FUNCTION_BLOCK AO1 (* Composite Function Block Type *)
  (* Standard: 61499-2 *)
  (* Version 0.0, 2018-12-26, 4DIAC-IDE, 4DIAC-Consortium *)
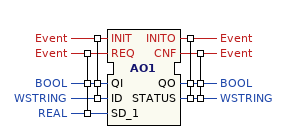
  EVENT_INPUT
    INIT WITH QI, ID; (* Initialization Request *)
    REQ WITH SD_1, QI; (* Normal Execution Request *)
  END_EVENT
  EVENT_OUTPUT
    INITO WITH QO, STATUS; (* Initialization Confirm *)
    CNF WITH QO, STATUS; (* Execution Confirmation *)
  END_EVENT
  VAR_INPUT
    QI : BOOL;
    ID : WSTRING;
    SD_1 : REAL;
  END_VAR
  VAR_OUTPUT
    QO : BOOL;
    STATUS : WSTRING;
  END_VAR
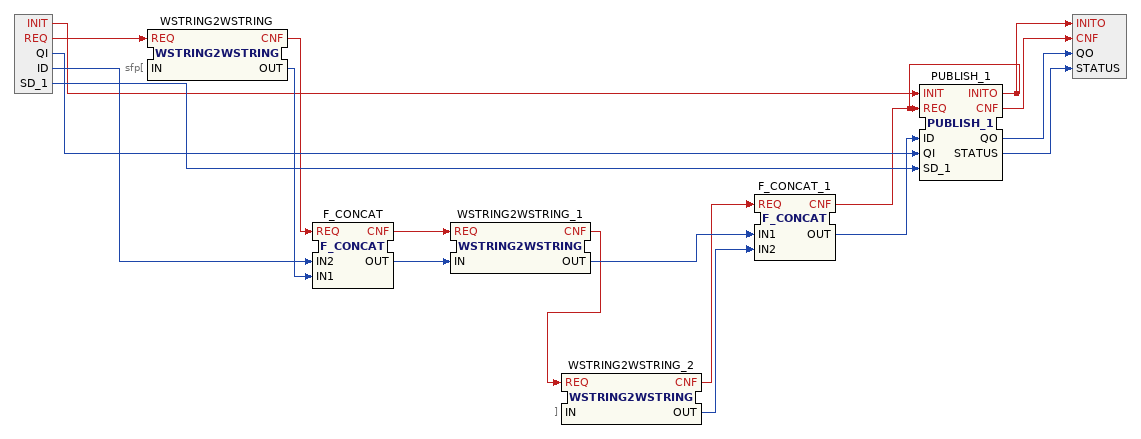
  FBS
    PUBLISH_1 : PUBLISH_1;
    F_CONCAT : F_CONCAT;
    WSTRING2WSTRING : WSTRING2WSTRING(IN := sfp[);
    WSTRING2WSTRING_1 : WSTRING2WSTRING;
    F_CONCAT_1 : F_CONCAT;
    WSTRING2WSTRING_2 : WSTRING2WSTRING(IN := ]);
  END_FBS
  EVENT_CONNECTIONS
    INIT TO PUBLISH_1.INIT;
    REQ TO WSTRING2WSTRING.REQ;
    WSTRING2WSTRING.CNF TO F_CONCAT.REQ;
    F_CONCAT.CNF TO WSTRING2WSTRING_1.REQ;
    WSTRING2WSTRING_2.CNF TO F_CONCAT_1.REQ;
    WSTRING2WSTRING_1.CNF TO WSTRING2WSTRING_2.REQ;
    F_CONCAT_1.CNF TO PUBLISH_1.REQ;
    PUBLISH_1.INITO TO INITO;
    PUBLISH_1.CNF TO CNF;
    PUBLISH_1.INITO TO PUBLISH_1.REQ;
  END_CONNECTIONS
  DATA_CONNECTIONS
    ID TO F_CONCAT.IN2;
    WSTRING2WSTRING.OUT TO F_CONCAT.IN1;
    F_CONCAT.OUT TO WSTRING2WSTRING_1.IN;
    WSTRING2WSTRING_1.OUT TO F_CONCAT_1.IN1;
    WSTRING2WSTRING_2.OUT TO F_CONCAT_1.IN2;
    F_CONCAT_1.OUT TO PUBLISH_1.ID;
    QI TO PUBLISH_1.QI;
    SD_1 TO PUBLISH_1.SD_1;
    PUBLISH_1.QO TO QO;
    PUBLISH_1.STATUS TO STATUS;
  END_CONNECTIONS
END_FUNCTION_BLOCK
